// TIA Portal V15.1 export
// export: Created 2024-05-17T05:38:39.8401583Z, ExportSetting WithDefaults, DisplayName Totally Integrated Automation Portal, DisplayVersion V15.1 Update 5, DisplayName TIA Portal Openness, DisplayVersion V15.1 Update 5, DisplayName SINAMICS Startdrive Advanced, DisplayVersion V15.1, DisplayName G130, G150, S120, S150, SINAMICS MV, S210, DisplayVersion V15.1, DisplayName G110M, G120, G120C, G120D, G120P, DisplayVersion V15.1, DisplayName STEP 7 Professional, DisplayVersion V15.1 Update 5, DisplayName STEP 7 Safety, DisplayVersion V15.1, DisplayName WinCC Professional, DisplayVersion V15.1 Update 5, DisplayName SIMATIC Visualization Architect, DisplayVersion V15.1
FUNCTION_BLOCK "LGBBitShift"   // FB6690, FBD
TITLE = LGBBitShift
{ S7_Optimized_Access := 'TRUE' }
VERSION : 0.1
// stored: AutoNumber false, IsIECCheckEnabled false, IsRetainMemResEnabled false, MemoryReserve 100, SetENOAutomatically False, UDAEnableTagReadback false
   VAR_INPUT
      I_ArrivedToPrev1 { ExternalAccessible := 'False'; ExternalVisible := 'False'; ExternalWritable := 'False'} : Bool;   // Arrived signal to previous transfer 1
      I_Bits1 { ExternalAccessible := 'False'; ExternalVisible := 'False'; ExternalWritable := 'False'} : Word;   // Bits transfer 1
      I_ArrivedToPrev2 { ExternalAccessible := 'False'; ExternalVisible := 'False'; ExternalWritable := 'False'} : Bool;   // Arrived signal to previous transfer 2
      I_Bits2 { ExternalAccessible := 'False'; ExternalVisible := 'False'; ExternalWritable := 'False'} : Word;   // Bits transfer 2
      I_ArrivedToPrev3 { ExternalAccessible := 'False'; ExternalVisible := 'False'; ExternalWritable := 'False'} : Bool;   // Arrived signal to previous transfer 3
      I_Bits3 { ExternalAccessible := 'False'; ExternalVisible := 'False'; ExternalWritable := 'False'} : Word;   // Bits transfer 3
      I_ArrivedToPrev4 { ExternalAccessible := 'False'; ExternalVisible := 'False'; ExternalWritable := 'False'} : Bool;   // Arrived signal to previous transfer 4
      I_Bits4 { ExternalAccessible := 'False'; ExternalVisible := 'False'; ExternalWritable := 'False'} : Word;   // Bits transfer 4
      I_NextShiftDone { ExternalAccessible := 'False'; ExternalVisible := 'False'; ExternalWritable := 'False'} : Bool;   // Shift to next position is done
   END_VAR
   VAR_OUTPUT
      O_ShiftDone1 { ExternalAccessible := 'False'; ExternalVisible := 'False'; ExternalWritable := 'False'} : Bool;   // Shift done transfer 1
      O_ShiftDone2 { ExternalAccessible := 'False'; ExternalVisible := 'False'; ExternalWritable := 'False'} : Bool;   // Shift done transfer 2
      O_ShiftDone3 { ExternalAccessible := 'False'; ExternalVisible := 'False'; ExternalWritable := 'False'} : Bool;   // Shift done transfer 3
      O_ShiftDone4 { ExternalAccessible := 'False'; ExternalVisible := 'False'; ExternalWritable := 'False'} : Bool;   // Shift done transfer 4
      O_Bits { ExternalAccessible := 'False'; ExternalVisible := 'False'; ExternalWritable := 'False'} : Int;   // Bits for this position
      O_Bit0 { ExternalAccessible := 'False'; ExternalVisible := 'False'; ExternalWritable := 'False'} : Bool;   // Bit 0
      O_Bit1 { ExternalAccessible := 'False'; ExternalVisible := 'False'; ExternalWritable := 'False'} : Bool;   // Bit 1
      O_Bit2 { ExternalAccessible := 'False'; ExternalVisible := 'False'; ExternalWritable := 'False'} : Bool;   // Bit 2
      O_Bit3 { ExternalAccessible := 'False'; ExternalVisible := 'False'; ExternalWritable := 'False'} : Bool;   // Bit 3
      O_Bit4 { ExternalAccessible := 'False'; ExternalVisible := 'False'; ExternalWritable := 'False'} : Bool;   // Bit 4
      O_Bit5 { ExternalAccessible := 'False'; ExternalVisible := 'False'; ExternalWritable := 'False'} : Bool;   // Bit 5
      O_Bit6 { ExternalAccessible := 'False'; ExternalVisible := 'False'; ExternalWritable := 'False'} : Bool;   // Bit 6
      O_Bit7 { ExternalAccessible := 'False'; ExternalVisible := 'False'; ExternalWritable := 'False'} : Bool;   // Bit 7
      O_Bit8 { ExternalAccessible := 'False'; ExternalVisible := 'False'; ExternalWritable := 'False'} : Bool;   // Bit 8
      O_Bit9 { ExternalAccessible := 'False'; ExternalVisible := 'False'; ExternalWritable := 'False'} : Bool;   // Bit 9
      O_Bit10 { ExternalAccessible := 'False'; ExternalVisible := 'False'; ExternalWritable := 'False'} : Bool;   // Bit 10
      O_Bit11 { ExternalAccessible := 'False'; ExternalVisible := 'False'; ExternalWritable := 'False'} : Bool;   // Bit 11
      O_Bit12 { ExternalAccessible := 'False'; ExternalVisible := 'False'; ExternalWritable := 'False'} : Bool;   // Bit 12
      O_Bit13 { ExternalAccessible := 'False'; ExternalVisible := 'False'; ExternalWritable := 'False'} : Bool;   // Bit 13
      O_Bit14 { ExternalAccessible := 'False'; ExternalVisible := 'False'; ExternalWritable := 'False'} : Bool;   // Bit 14
      O_Bit15 { ExternalAccessible := 'False'; ExternalVisible := 'False'; ExternalWritable := 'False'} : Bool;   // Bit 15
      O_AlarmABCondition { ExternalAccessible := 'False'; ExternalVisible := 'False'; ExternalWritable := 'False'} : Bool;   // Alarm AB Condition
      O_AlarmA { ExternalAccessible := 'False'; ExternalVisible := 'False'; ExternalWritable := 'False'} : Bool;   // Alarm A
      O_AlarmB { ExternalAccessible := 'False'; ExternalVisible := 'False'; ExternalWritable := 'False'} : Bool;   // Alarm B
      O_AlarmC { ExternalAccessible := 'False'; ExternalVisible := 'False'; ExternalWritable := 'False'} : Bool;   // Alarm C
      O_AlarmD { ExternalAccessible := 'False'; ExternalVisible := 'False'; ExternalWritable := 'False'} : Bool;   // Alarm D
      H_AlarmDWord { ExternalAccessible := 'False'; ExternalVisible := 'False'; ExternalWritable := 'False'} : DWord;   // HMI Animation
   END_VAR
   VAR_IN_OUT
      IO_Modes : "Modes";   // Modes
      H_HMI : "H_HMI";   // Icon Animation
      H_GBBitShift : "H_GBBitShift";   // Animation
      C_Config : "BitShiftConfig";   // Config
   END_VAR
   VAR
      AC_NoBitShift { ExternalAccessible := 'False'; ExternalVisible := 'False'; ExternalWritable := 'False'} : Bool;   // Alarm No Bit Shift
      PulseArrivedToPrev1 { ExternalAccessible := 'False'; ExternalVisible := 'False'; ExternalWritable := 'False'} : Bool;   // Pulse Arrived Signal to Previous Transfer 1
      Arrived1 { ExternalAccessible := 'False'; ExternalVisible := 'False'; ExternalWritable := 'False'} : Bool;   // Arrived 1
      PulseArrivedToPrev2 { ExternalAccessible := 'False'; ExternalVisible := 'False'; ExternalWritable := 'False'} : Bool;   // Pulse Arrived Signal to Previous Transfer 2
      Arrived2 { ExternalAccessible := 'False'; ExternalVisible := 'False'; ExternalWritable := 'False'} : Bool;   // Arrived 2
      PulseArrivedToPrev3 { ExternalAccessible := 'False'; ExternalVisible := 'False'; ExternalWritable := 'False'} : Bool;   // Pulse Arrived Signal to Previous Transfer 3
      Arrived3 { ExternalAccessible := 'False'; ExternalVisible := 'False'; ExternalWritable := 'False'} : Bool;   // Arrived 3
      PulseArrivedToPrev4 { ExternalAccessible := 'False'; ExternalVisible := 'False'; ExternalWritable := 'False'} : Bool;   // Pulse Arrived Signal to Previous Transfer 4
      Arrived4 { ExternalAccessible := 'False'; ExternalVisible := 'False'; ExternalWritable := 'False'} : Bool;   // Arrived 4
   END_VAR
   VAR RETAIN
      Bits { ExternalAccessible := 'False'; ExternalVisible := 'False'; ExternalWritable := 'False'} : Word;   // Bits of this position
   END_VAR
   VAR
      AlarmA { ExternalAccessible := 'False'; ExternalVisible := 'False'; ExternalWritable := 'False'} : Bool;   // Alarm A
      AlarmB { ExternalAccessible := 'False'; ExternalVisible := 'False'; ExternalWritable := 'False'} : Bool;   // Alarm B
      AlarmC { ExternalAccessible := 'False'; ExternalVisible := 'False'; ExternalWritable := 'False'} : Bool;   // Alarm C
      AlarmD { ExternalAccessible := 'False'; ExternalVisible := 'False'; ExternalWritable := 'False'} : Bool;   // Alarm D
      AlarmABCondition { ExternalAccessible := 'False'; ExternalVisible := 'False'; ExternalWritable := 'False'} : Bool;   // Alarm AB Condition
   END_VAR
   VAR_TEMP   // added for the SCL form of the ladder/FBD networks
      _w1 : Bool;
   END_VAR
BEGIN

REGION Network 1: **** 4.4 - Machine status - Calculated **** Pulse Arrived Signal 1 To previous
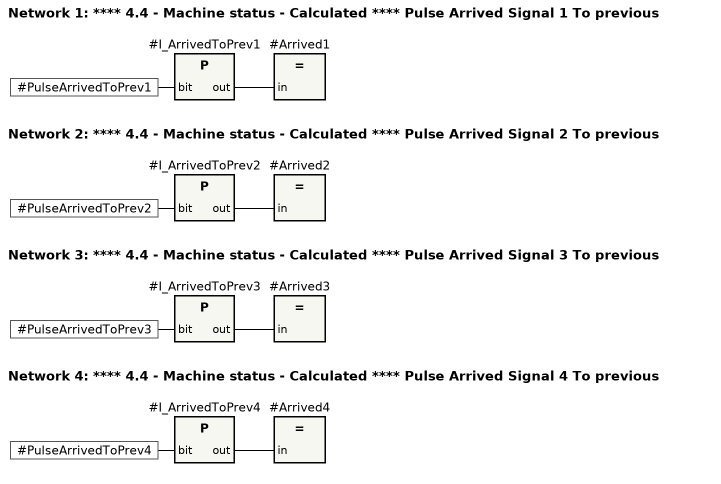
   #_w1 := #I_ArrivedToPrev1 AND NOT #PulseArrivedToPrev1;   // rising edge of #I_ArrivedToPrev1
   #PulseArrivedToPrev1 := #I_ArrivedToPrev1;
   #Arrived1 := #_w1;
END_REGION

REGION Network 2: **** 4.4 - Machine status - Calculated **** Pulse Arrived Signal 2 To previous
   #_w1 := #I_ArrivedToPrev2 AND NOT #PulseArrivedToPrev2;   // rising edge of #I_ArrivedToPrev2
   #PulseArrivedToPrev2 := #I_ArrivedToPrev2;
   #Arrived2 := #_w1;
END_REGION

REGION Network 3: **** 4.4 - Machine status - Calculated **** Pulse Arrived Signal 3 To previous
   #_w1 := #I_ArrivedToPrev3 AND NOT #PulseArrivedToPrev3;   // rising edge of #I_ArrivedToPrev3
   #PulseArrivedToPrev3 := #I_ArrivedToPrev3;
   #Arrived3 := #_w1;
END_REGION

REGION Network 4: **** 4.4 - Machine status - Calculated **** Pulse Arrived Signal 4 To previous
   #_w1 := #I_ArrivedToPrev4 AND NOT #PulseArrivedToPrev4;   // rising edge of #I_ArrivedToPrev4
   #PulseArrivedToPrev4 := #I_ArrivedToPrev4;
   #Arrived4 := #_w1;
END_REGION

REGION Network 5: **** 4.4 - Machine status - Calculated **** Copy Bits from Transfer 1
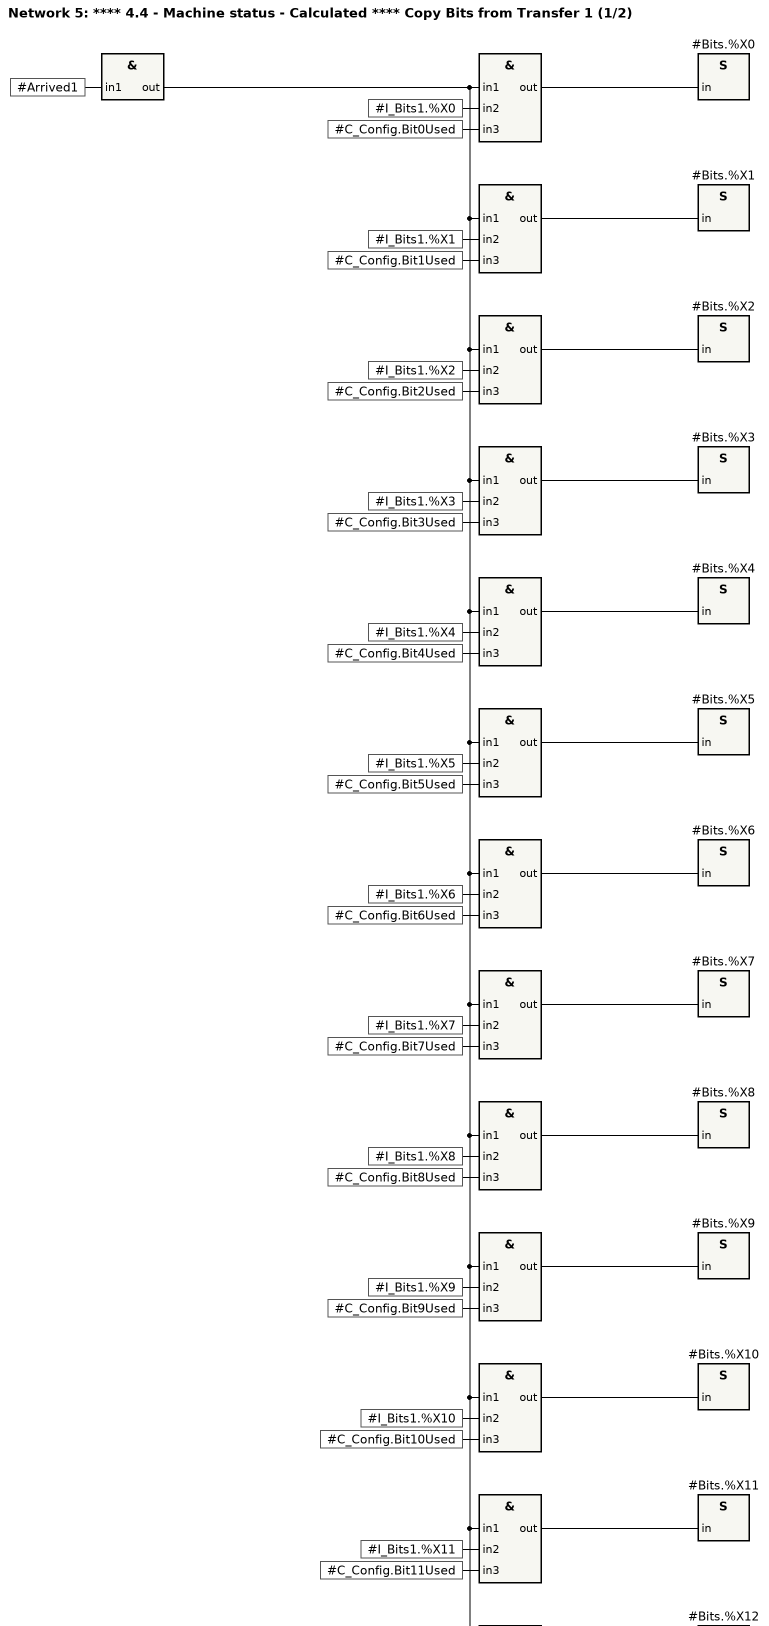
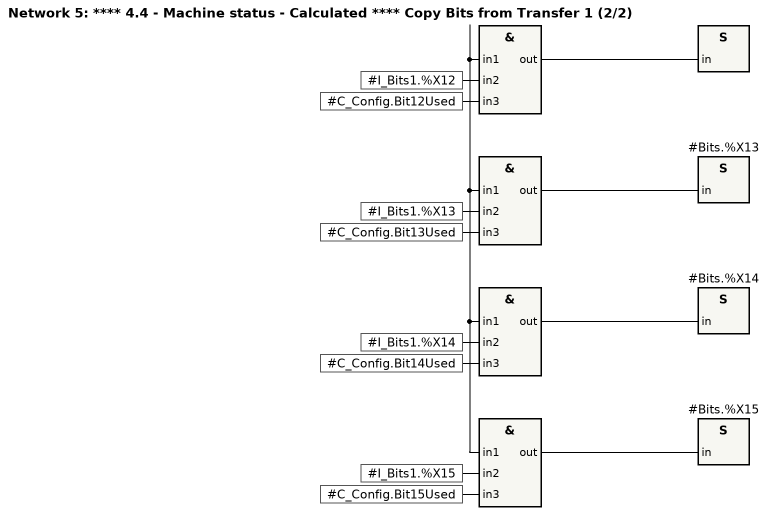
   IF #Arrived1 AND #I_Bits1.%X0 AND #C_Config.Bit0Used THEN #Bits.%X0 := TRUE; END_IF;
   IF #Arrived1 AND #I_Bits1.%X1 AND #C_Config.Bit1Used THEN #Bits.%X1 := TRUE; END_IF;
   IF #Arrived1 AND #I_Bits1.%X2 AND #C_Config.Bit2Used THEN #Bits.%X2 := TRUE; END_IF;
   IF #Arrived1 AND #I_Bits1.%X3 AND #C_Config.Bit3Used THEN #Bits.%X3 := TRUE; END_IF;
   IF #Arrived1 AND #I_Bits1.%X4 AND #C_Config.Bit4Used THEN #Bits.%X4 := TRUE; END_IF;
   IF #Arrived1 AND #I_Bits1.%X5 AND #C_Config.Bit5Used THEN #Bits.%X5 := TRUE; END_IF;
   IF #Arrived1 AND #I_Bits1.%X6 AND #C_Config.Bit6Used THEN #Bits.%X6 := TRUE; END_IF;
   IF #Arrived1 AND #I_Bits1.%X7 AND #C_Config.Bit7Used THEN #Bits.%X7 := TRUE; END_IF;
   IF #Arrived1 AND #I_Bits1.%X8 AND #C_Config.Bit8Used THEN #Bits.%X8 := TRUE; END_IF;
   IF #Arrived1 AND #I_Bits1.%X9 AND #C_Config.Bit9Used THEN #Bits.%X9 := TRUE; END_IF;
   IF #Arrived1 AND #I_Bits1.%X10 AND #C_Config.Bit10Used THEN #Bits.%X10 := TRUE; END_IF;
   IF #Arrived1 AND #I_Bits1.%X11 AND #C_Config.Bit11Used THEN #Bits.%X11 := TRUE; END_IF;
   IF #Arrived1 AND #I_Bits1.%X12 AND #C_Config.Bit12Used THEN #Bits.%X12 := TRUE; END_IF;
   IF #Arrived1 AND #I_Bits1.%X13 AND #C_Config.Bit13Used THEN #Bits.%X13 := TRUE; END_IF;
   IF #Arrived1 AND #I_Bits1.%X14 AND #C_Config.Bit14Used THEN #Bits.%X14 := TRUE; END_IF;
   IF #Arrived1 AND #I_Bits1.%X15 AND #C_Config.Bit15Used THEN #Bits.%X15 := TRUE; END_IF;
END_REGION

REGION Network 6: **** 4.4 - Machine status - Calculated **** Copy Bits from Transfer 2
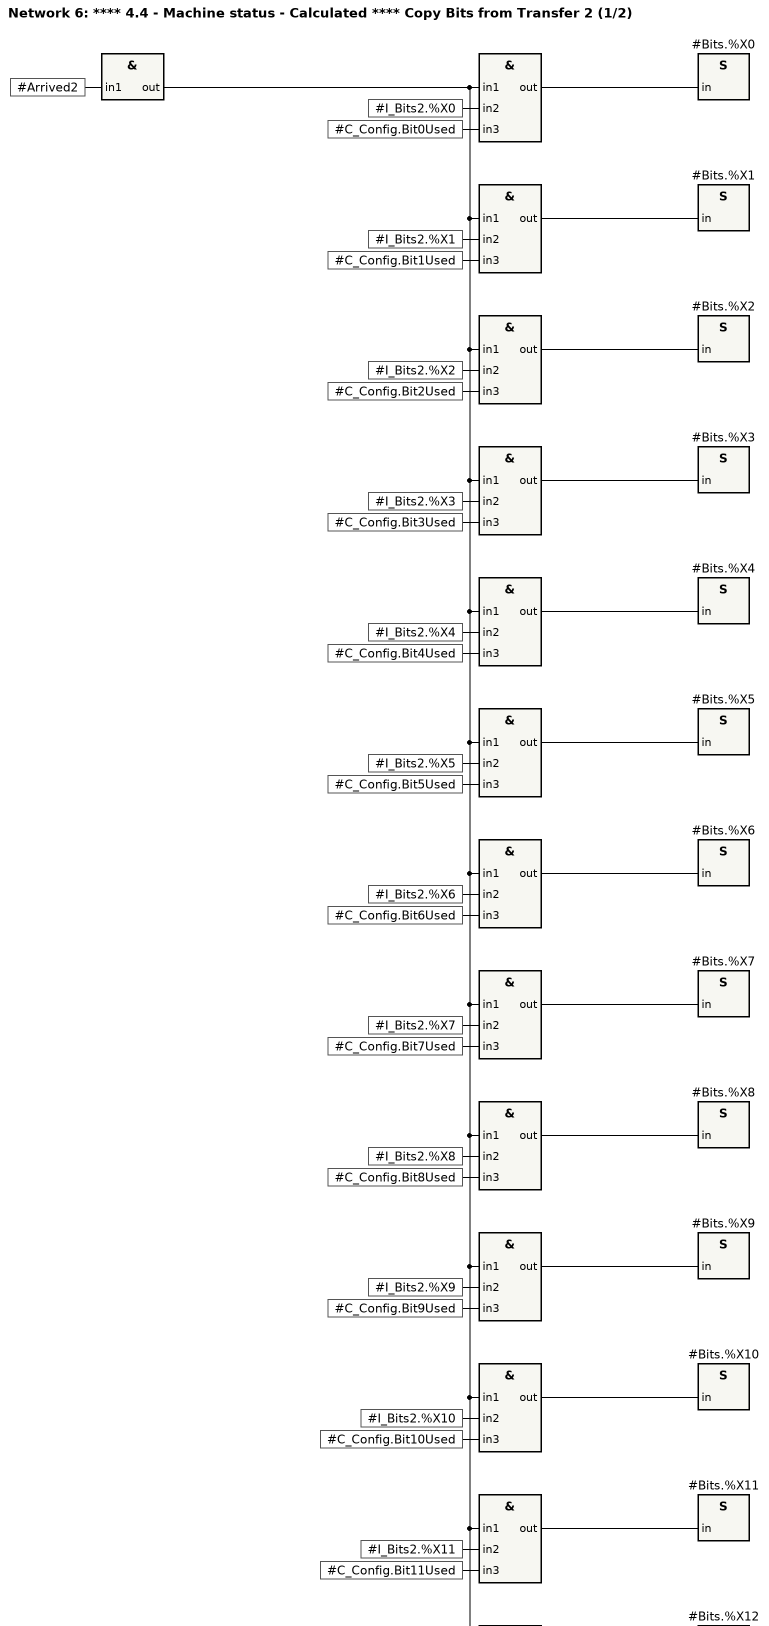
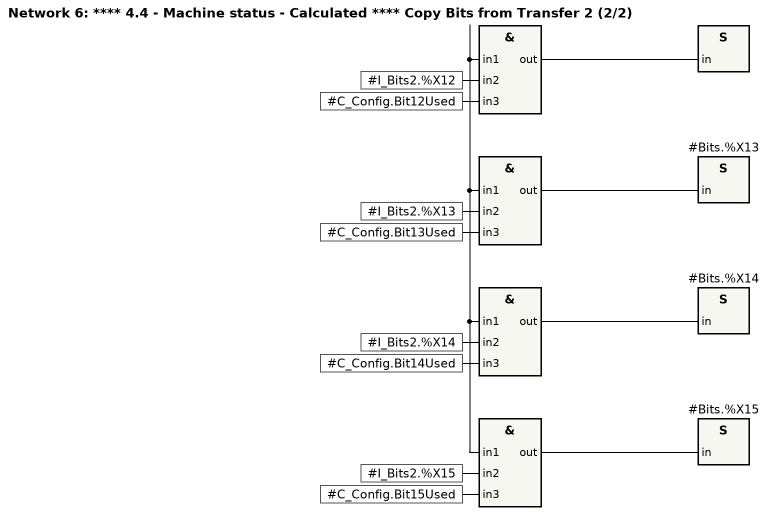
   IF #Arrived2 AND #I_Bits2.%X0 AND #C_Config.Bit0Used THEN #Bits.%X0 := TRUE; END_IF;
   IF #Arrived2 AND #I_Bits2.%X1 AND #C_Config.Bit1Used THEN #Bits.%X1 := TRUE; END_IF;
   IF #Arrived2 AND #I_Bits2.%X2 AND #C_Config.Bit2Used THEN #Bits.%X2 := TRUE; END_IF;
   IF #Arrived2 AND #I_Bits2.%X3 AND #C_Config.Bit3Used THEN #Bits.%X3 := TRUE; END_IF;
   IF #Arrived2 AND #I_Bits2.%X4 AND #C_Config.Bit4Used THEN #Bits.%X4 := TRUE; END_IF;
   IF #Arrived2 AND #I_Bits2.%X5 AND #C_Config.Bit5Used THEN #Bits.%X5 := TRUE; END_IF;
   IF #Arrived2 AND #I_Bits2.%X6 AND #C_Config.Bit6Used THEN #Bits.%X6 := TRUE; END_IF;
   IF #Arrived2 AND #I_Bits2.%X7 AND #C_Config.Bit7Used THEN #Bits.%X7 := TRUE; END_IF;
   IF #Arrived2 AND #I_Bits2.%X8 AND #C_Config.Bit8Used THEN #Bits.%X8 := TRUE; END_IF;
   IF #Arrived2 AND #I_Bits2.%X9 AND #C_Config.Bit9Used THEN #Bits.%X9 := TRUE; END_IF;
   IF #Arrived2 AND #I_Bits2.%X10 AND #C_Config.Bit10Used THEN #Bits.%X10 := TRUE; END_IF;
   IF #Arrived2 AND #I_Bits2.%X11 AND #C_Config.Bit11Used THEN #Bits.%X11 := TRUE; END_IF;
   IF #Arrived2 AND #I_Bits2.%X12 AND #C_Config.Bit12Used THEN #Bits.%X12 := TRUE; END_IF;
   IF #Arrived2 AND #I_Bits2.%X13 AND #C_Config.Bit13Used THEN #Bits.%X13 := TRUE; END_IF;
   IF #Arrived2 AND #I_Bits2.%X14 AND #C_Config.Bit14Used THEN #Bits.%X14 := TRUE; END_IF;
   IF #Arrived2 AND #I_Bits2.%X15 AND #C_Config.Bit15Used THEN #Bits.%X15 := TRUE; END_IF;
END_REGION

REGION Network 7: **** 4.4 - Machine status - Calculated **** Copy Bits from Transfer 3
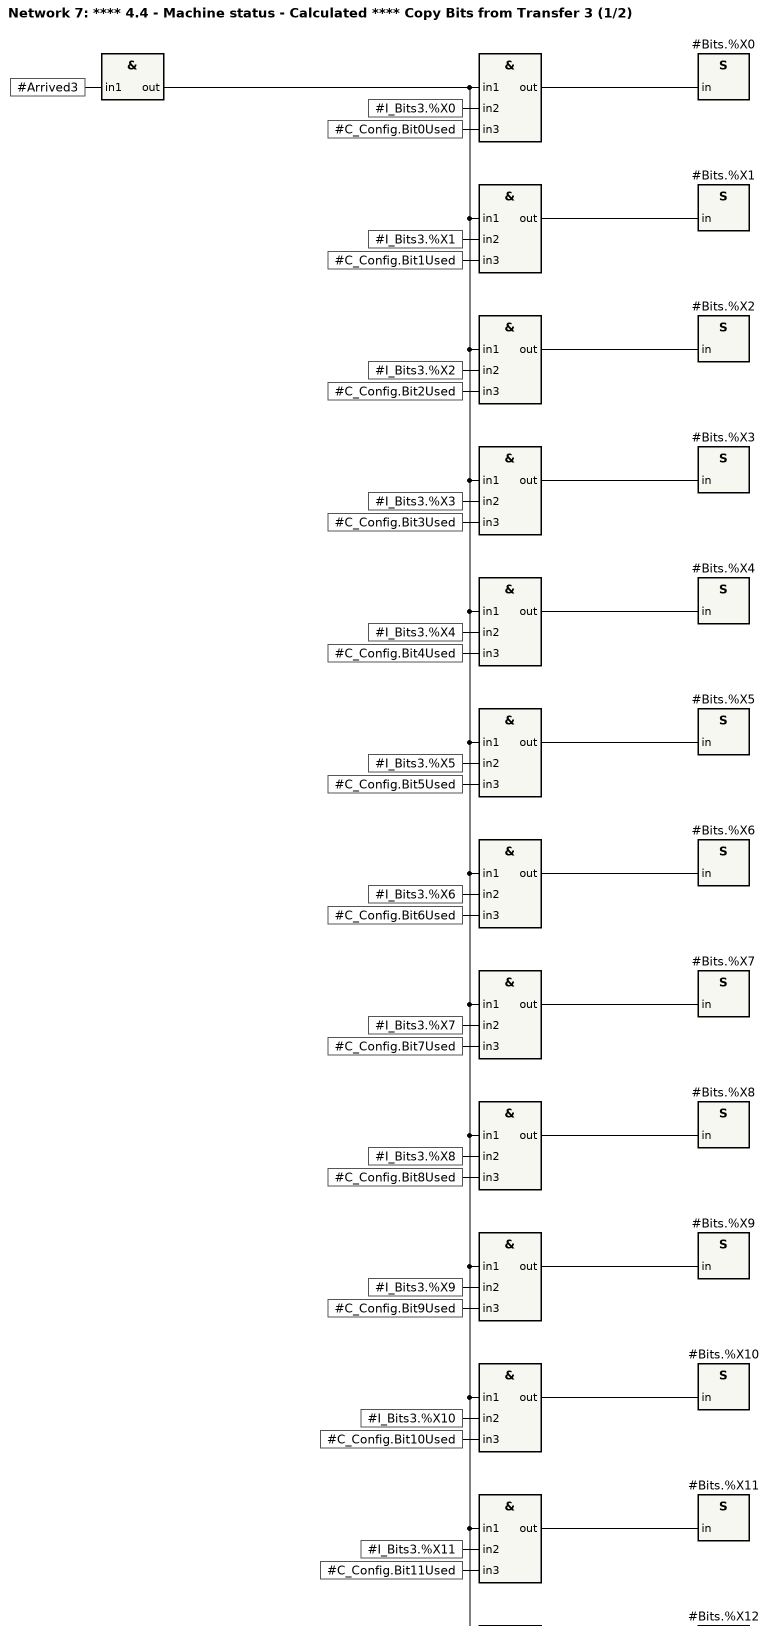
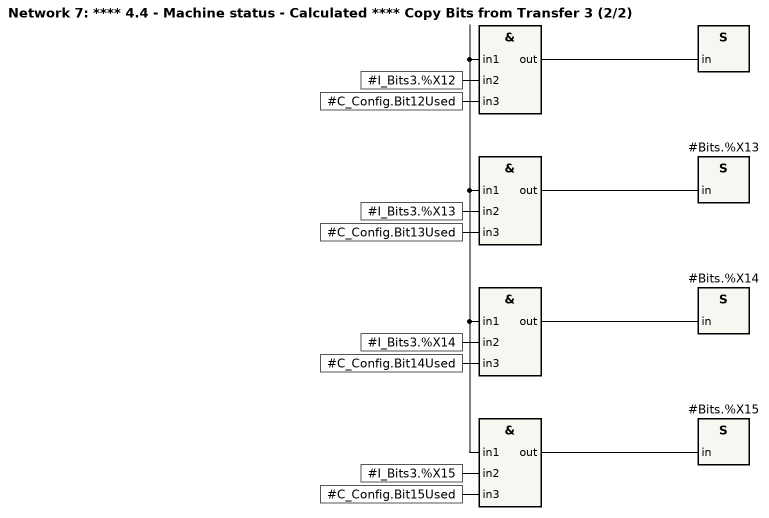
   IF #Arrived3 AND #I_Bits3.%X0 AND #C_Config.Bit0Used THEN #Bits.%X0 := TRUE; END_IF;
   IF #Arrived3 AND #I_Bits3.%X1 AND #C_Config.Bit1Used THEN #Bits.%X1 := TRUE; END_IF;
   IF #Arrived3 AND #I_Bits3.%X2 AND #C_Config.Bit2Used THEN #Bits.%X2 := TRUE; END_IF;
   IF #Arrived3 AND #I_Bits3.%X3 AND #C_Config.Bit3Used THEN #Bits.%X3 := TRUE; END_IF;
   IF #Arrived3 AND #I_Bits3.%X4 AND #C_Config.Bit4Used THEN #Bits.%X4 := TRUE; END_IF;
   IF #Arrived3 AND #I_Bits3.%X5 AND #C_Config.Bit5Used THEN #Bits.%X5 := TRUE; END_IF;
   IF #Arrived3 AND #I_Bits3.%X6 AND #C_Config.Bit6Used THEN #Bits.%X6 := TRUE; END_IF;
   IF #Arrived3 AND #I_Bits3.%X7 AND #C_Config.Bit7Used THEN #Bits.%X7 := TRUE; END_IF;
   IF #Arrived3 AND #I_Bits3.%X8 AND #C_Config.Bit8Used THEN #Bits.%X8 := TRUE; END_IF;
   IF #Arrived3 AND #I_Bits3.%X9 AND #C_Config.Bit9Used THEN #Bits.%X9 := TRUE; END_IF;
   IF #Arrived3 AND #I_Bits3.%X10 AND #C_Config.Bit10Used THEN #Bits.%X10 := TRUE; END_IF;
   IF #Arrived3 AND #I_Bits3.%X11 AND #C_Config.Bit11Used THEN #Bits.%X11 := TRUE; END_IF;
   IF #Arrived3 AND #I_Bits3.%X12 AND #C_Config.Bit12Used THEN #Bits.%X12 := TRUE; END_IF;
   IF #Arrived3 AND #I_Bits3.%X13 AND #C_Config.Bit13Used THEN #Bits.%X13 := TRUE; END_IF;
   IF #Arrived3 AND #I_Bits3.%X14 AND #C_Config.Bit14Used THEN #Bits.%X14 := TRUE; END_IF;
   IF #Arrived3 AND #I_Bits3.%X15 AND #C_Config.Bit15Used THEN #Bits.%X15 := TRUE; END_IF;
END_REGION

REGION Network 8: **** 4.4 - Machine status - Calculated **** Copy Bits from Transfer 4
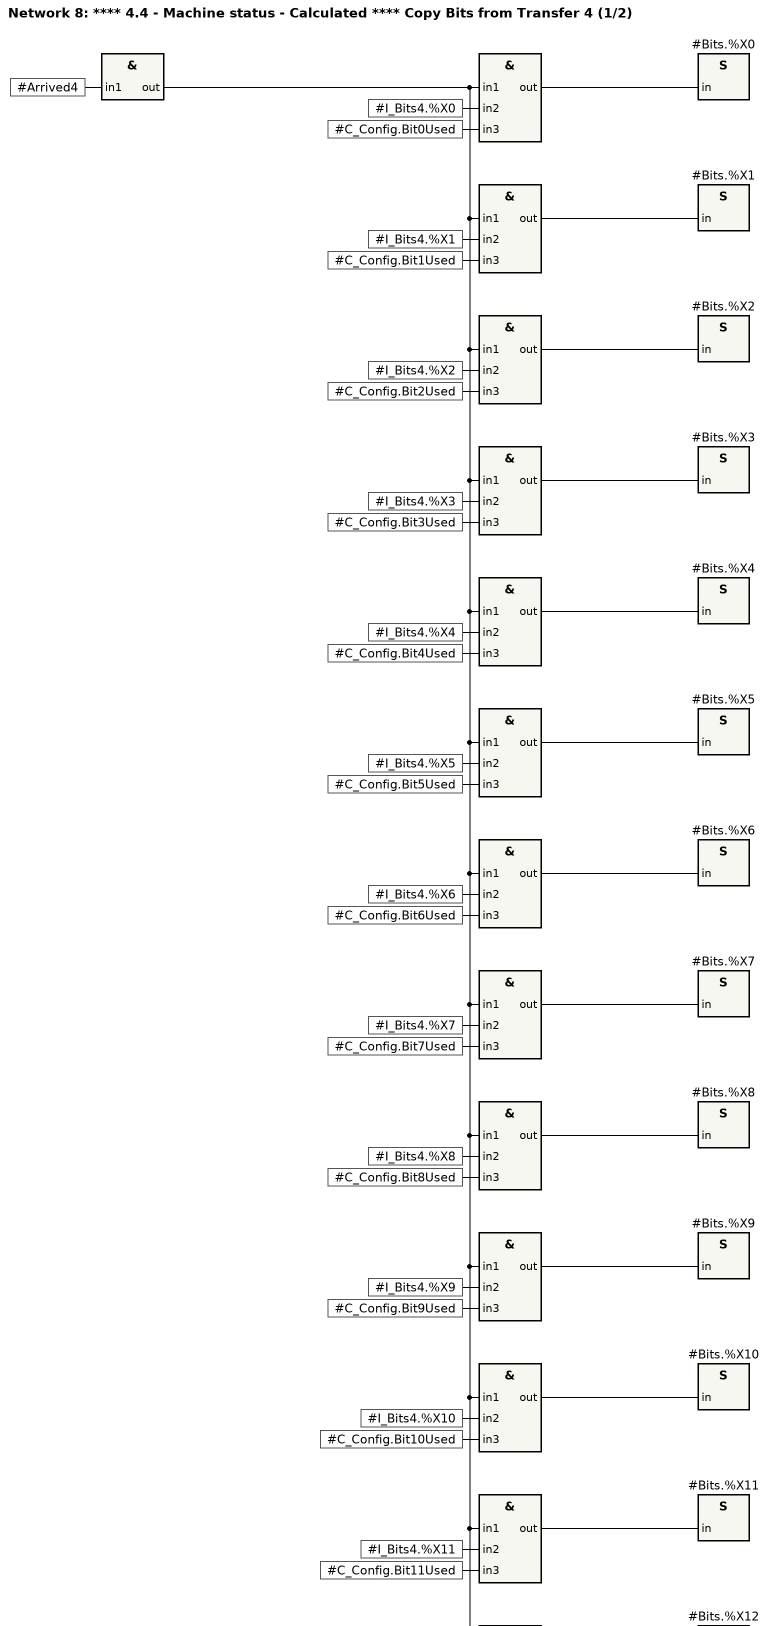
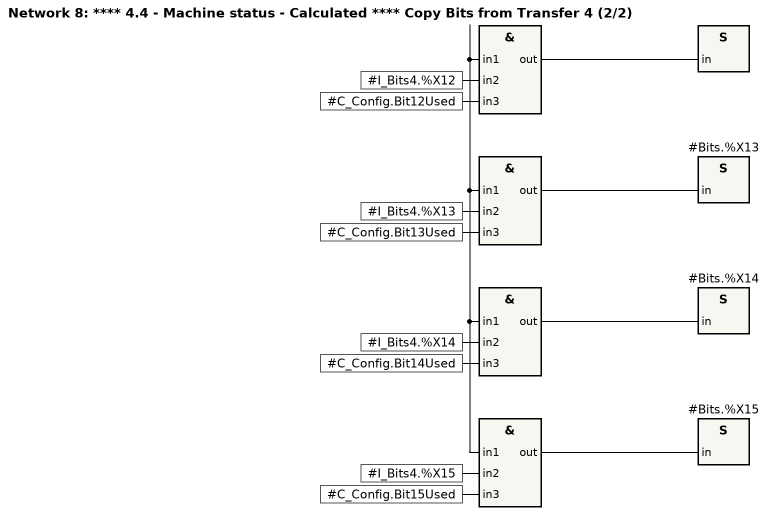
   IF #Arrived4 AND #I_Bits4.%X0 AND #C_Config.Bit0Used THEN #Bits.%X0 := TRUE; END_IF;
   IF #Arrived4 AND #I_Bits4.%X1 AND #C_Config.Bit1Used THEN #Bits.%X1 := TRUE; END_IF;
   IF #Arrived4 AND #I_Bits4.%X2 AND #C_Config.Bit2Used THEN #Bits.%X2 := TRUE; END_IF;
   IF #Arrived4 AND #I_Bits4.%X3 AND #C_Config.Bit3Used THEN #Bits.%X3 := TRUE; END_IF;
   IF #Arrived4 AND #I_Bits4.%X4 AND #C_Config.Bit4Used THEN #Bits.%X4 := TRUE; END_IF;
   IF #Arrived4 AND #I_Bits4.%X5 AND #C_Config.Bit5Used THEN #Bits.%X5 := TRUE; END_IF;
   IF #Arrived4 AND #I_Bits4.%X6 AND #C_Config.Bit6Used THEN #Bits.%X6 := TRUE; END_IF;
   IF #Arrived4 AND #I_Bits4.%X7 AND #C_Config.Bit7Used THEN #Bits.%X7 := TRUE; END_IF;
   IF #Arrived4 AND #I_Bits4.%X8 AND #C_Config.Bit8Used THEN #Bits.%X8 := TRUE; END_IF;
   IF #Arrived4 AND #I_Bits4.%X9 AND #C_Config.Bit9Used THEN #Bits.%X9 := TRUE; END_IF;
   IF #Arrived4 AND #I_Bits4.%X10 AND #C_Config.Bit10Used THEN #Bits.%X10 := TRUE; END_IF;
   IF #Arrived4 AND #I_Bits4.%X11 AND #C_Config.Bit11Used THEN #Bits.%X11 := TRUE; END_IF;
   IF #Arrived4 AND #I_Bits4.%X12 AND #C_Config.Bit12Used THEN #Bits.%X12 := TRUE; END_IF;
   IF #Arrived4 AND #I_Bits4.%X13 AND #C_Config.Bit13Used THEN #Bits.%X13 := TRUE; END_IF;
   IF #Arrived4 AND #I_Bits4.%X14 AND #C_Config.Bit14Used THEN #Bits.%X14 := TRUE; END_IF;
   IF #Arrived4 AND #I_Bits4.%X15 AND #C_Config.Bit15Used THEN #Bits.%X15 := TRUE; END_IF;
END_REGION

REGION Network 9: **** 4.4 - Machine status - Calculated **** Reset Data when shift to the next position is done
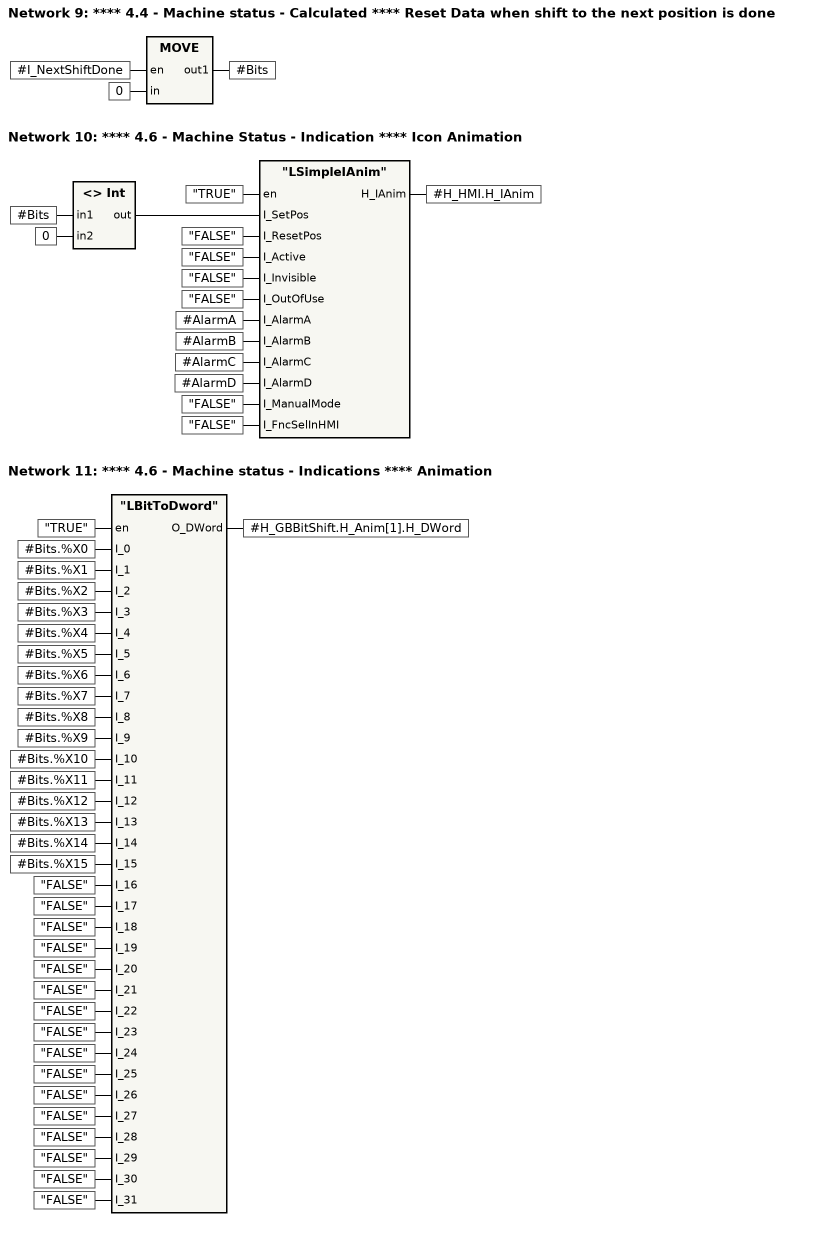
   IF #I_NextShiftDone THEN #Bits := 0; END_IF;
END_REGION

REGION Network 10: **** 4.6 - Machine Status - Indication **** Icon Animation
   IF "TRUE" THEN
       "LSimpleIAnim"(I_SetPos := #Bits <> 0,
                      I_ResetPos := "FALSE",
                      I_Active := "FALSE",
                      I_Invisible := "FALSE",
                      I_OutOfUse := "FALSE",
                      I_AlarmA := #AlarmA,
                      I_AlarmB := #AlarmB,
                      I_AlarmC := #AlarmC,
                      I_AlarmD := #AlarmD,
                      I_ManualMode := "FALSE",
                      I_FncSelInHMI := "FALSE",
                      H_IAnim => #H_HMI.H_IAnim);
   END_IF;
END_REGION

REGION Network 11: **** 4.6 - Machine status - Indications **** Animation
   IF "TRUE" THEN
       "LBitToDword"(I_0 := #Bits.%X0,
                     I_1 := #Bits.%X1,
                     I_2 := #Bits.%X2,
                     I_3 := #Bits.%X3,
                     I_4 := #Bits.%X4,
                     I_5 := #Bits.%X5,
                     I_6 := #Bits.%X6,
                     I_7 := #Bits.%X7,
                     I_8 := #Bits.%X8,
                     I_9 := #Bits.%X9,
                     I_10 := #Bits.%X10,
                     I_11 := #Bits.%X11,
                     I_12 := #Bits.%X12,
                     I_13 := #Bits.%X13,
                     I_14 := #Bits.%X14,
                     I_15 := #Bits.%X15,
                     I_16 := "FALSE",
                     I_17 := "FALSE",
                     I_18 := "FALSE",
                     I_19 := "FALSE",
                     I_20 := "FALSE",
                     I_21 := "FALSE",
                     I_22 := "FALSE",
                     I_23 := "FALSE",
                     I_24 := "FALSE",
                     I_25 := "FALSE",
                     I_26 := "FALSE",
                     I_27 := "FALSE",
                     I_28 := "FALSE",
                     I_29 := "FALSE",
                     I_30 := "FALSE",
                     I_31 := "FALSE",
                     O_DWord => #H_GBBitShift.H_Anim[1].H_DWord);
   END_IF;
END_REGION

REGION Network 12: **** 4.6 - Machine status - Indications **** Animation
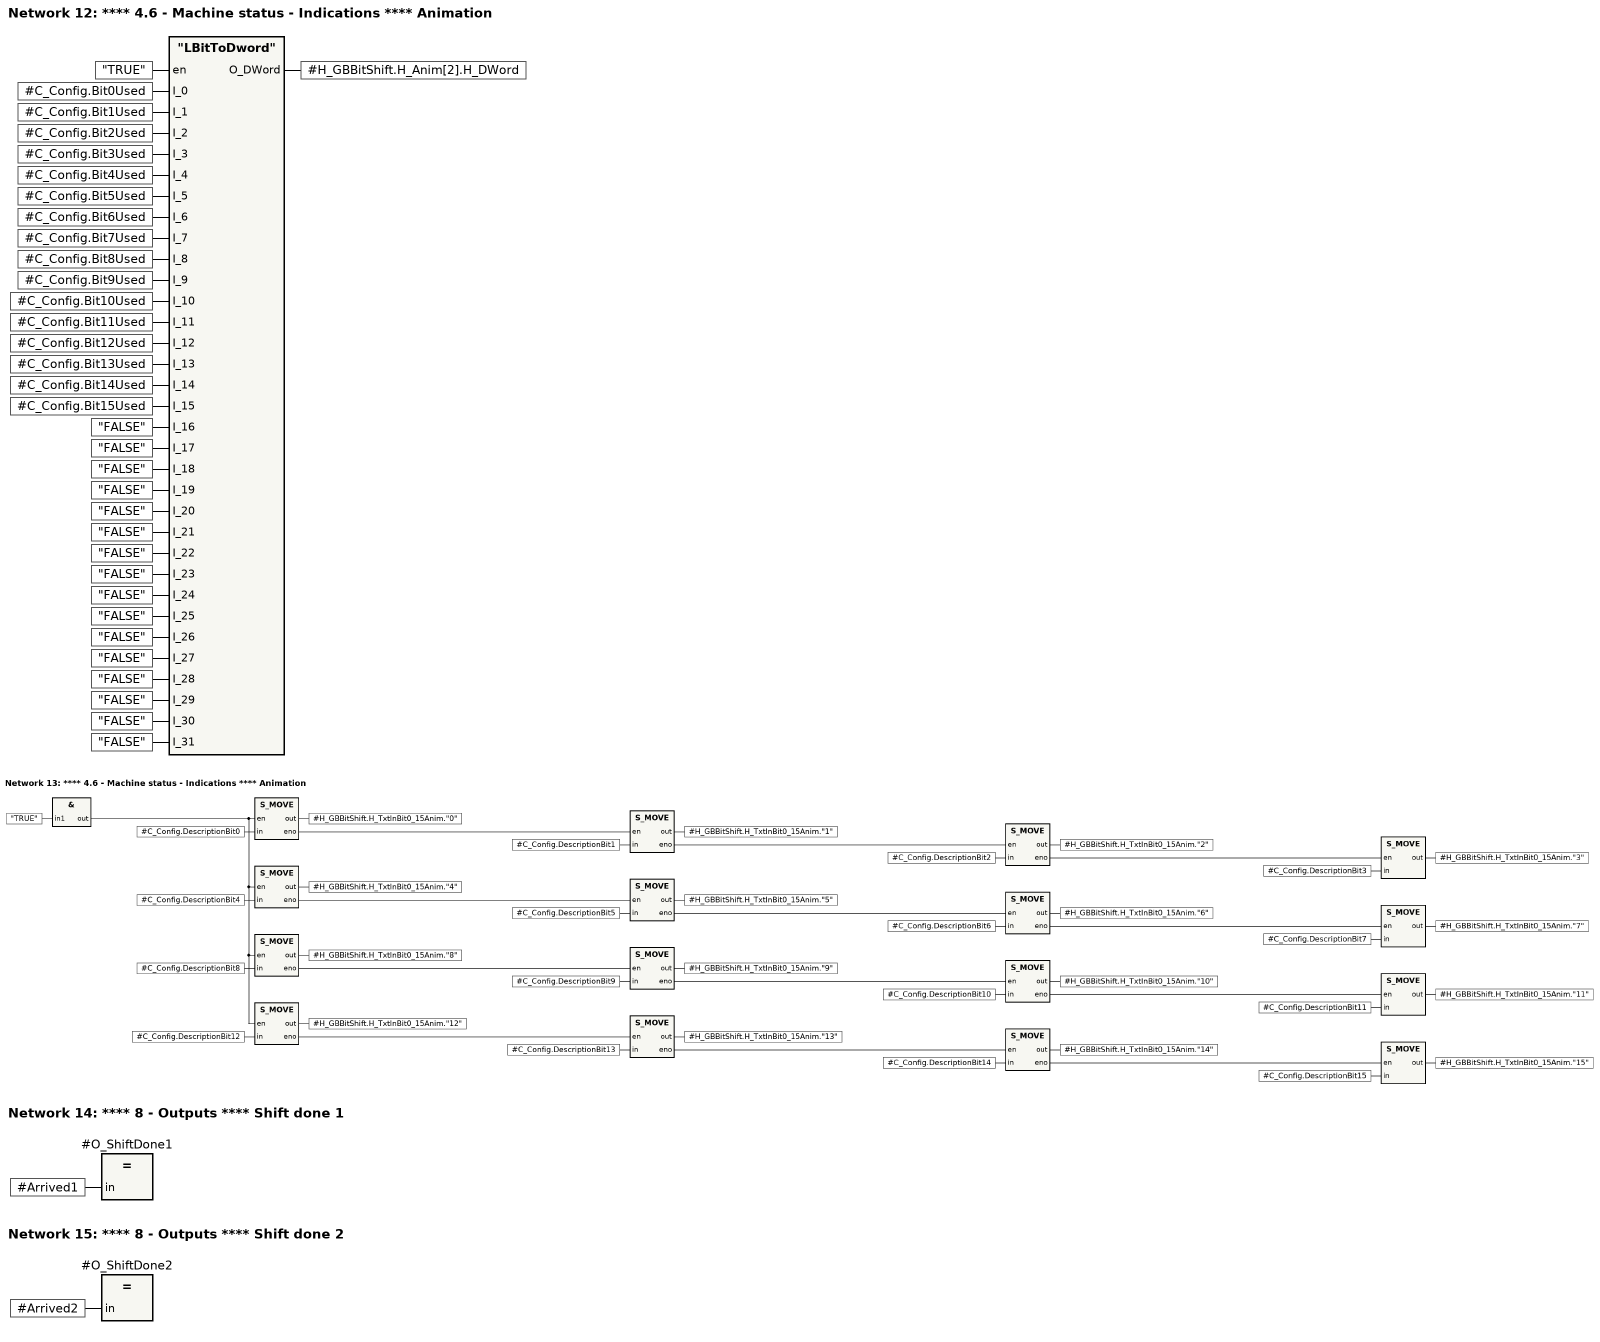
   IF "TRUE" THEN
       "LBitToDword"(I_0 := #C_Config.Bit0Used,
                     I_1 := #C_Config.Bit1Used,
                     I_2 := #C_Config.Bit2Used,
                     I_3 := #C_Config.Bit3Used,
                     I_4 := #C_Config.Bit4Used,
                     I_5 := #C_Config.Bit5Used,
                     I_6 := #C_Config.Bit6Used,
                     I_7 := #C_Config.Bit7Used,
                     I_8 := #C_Config.Bit8Used,
                     I_9 := #C_Config.Bit9Used,
                     I_10 := #C_Config.Bit10Used,
                     I_11 := #C_Config.Bit11Used,
                     I_12 := #C_Config.Bit12Used,
                     I_13 := #C_Config.Bit13Used,
                     I_14 := #C_Config.Bit14Used,
                     I_15 := #C_Config.Bit15Used,
                     I_16 := "FALSE",
                     I_17 := "FALSE",
                     I_18 := "FALSE",
                     I_19 := "FALSE",
                     I_20 := "FALSE",
                     I_21 := "FALSE",
                     I_22 := "FALSE",
                     I_23 := "FALSE",
                     I_24 := "FALSE",
                     I_25 := "FALSE",
                     I_26 := "FALSE",
                     I_27 := "FALSE",
                     I_28 := "FALSE",
                     I_29 := "FALSE",
                     I_30 := "FALSE",
                     I_31 := "FALSE",
                     O_DWord => #H_GBBitShift.H_Anim[2].H_DWord);
   END_IF;
END_REGION

REGION Network 13: **** 4.6 - Machine status - Indications **** Animation
   IF "TRUE" THEN
       #H_GBBitShift.H_TxtInBit0_15Anim."0" := #C_Config.DescriptionBit0;
       #H_GBBitShift.H_TxtInBit0_15Anim."1" := #C_Config.DescriptionBit1;
       #H_GBBitShift.H_TxtInBit0_15Anim."2" := #C_Config.DescriptionBit2;
       #H_GBBitShift.H_TxtInBit0_15Anim."3" := #C_Config.DescriptionBit3;
       #H_GBBitShift.H_TxtInBit0_15Anim."4" := #C_Config.DescriptionBit4;
       #H_GBBitShift.H_TxtInBit0_15Anim."5" := #C_Config.DescriptionBit5;
       #H_GBBitShift.H_TxtInBit0_15Anim."6" := #C_Config.DescriptionBit6;
       #H_GBBitShift.H_TxtInBit0_15Anim."7" := #C_Config.DescriptionBit7;
       #H_GBBitShift.H_TxtInBit0_15Anim."8" := #C_Config.DescriptionBit8;
       #H_GBBitShift.H_TxtInBit0_15Anim."9" := #C_Config.DescriptionBit9;
       #H_GBBitShift.H_TxtInBit0_15Anim."10" := #C_Config.DescriptionBit10;
       #H_GBBitShift.H_TxtInBit0_15Anim."11" := #C_Config.DescriptionBit11;
       #H_GBBitShift.H_TxtInBit0_15Anim."12" := #C_Config.DescriptionBit12;
       #H_GBBitShift.H_TxtInBit0_15Anim."13" := #C_Config.DescriptionBit13;
       #H_GBBitShift.H_TxtInBit0_15Anim."14" := #C_Config.DescriptionBit14;
       #H_GBBitShift.H_TxtInBit0_15Anim."15" := #C_Config.DescriptionBit15;
   END_IF;
END_REGION

REGION Network 14: **** 8 - Outputs **** Shift done 1
   #O_ShiftDone1 := #Arrived1;
END_REGION

REGION Network 15: **** 8 - Outputs **** Shift done 2
   #O_ShiftDone2 := #Arrived2;
END_REGION

REGION Network 16: **** 8 - Outputs **** Shift done 3
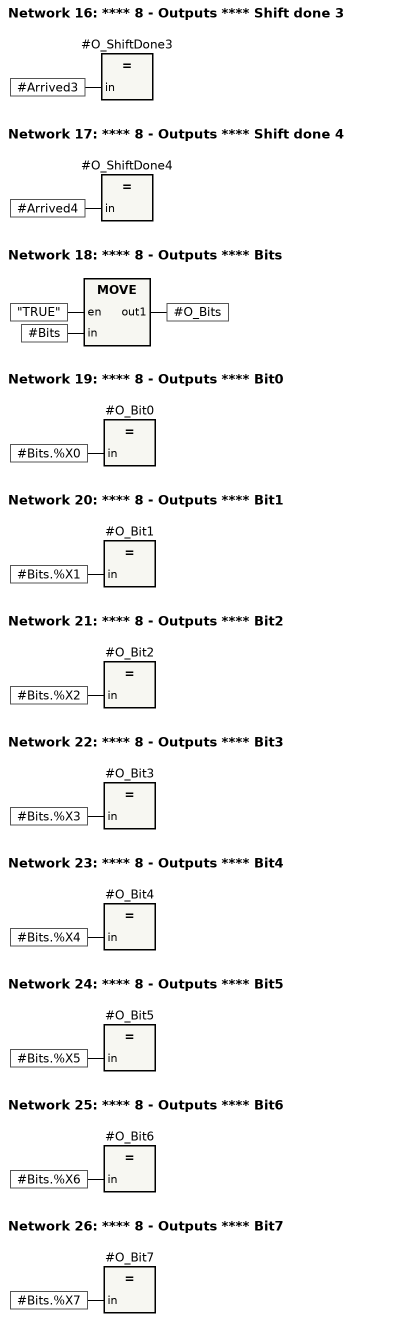
   #O_ShiftDone3 := #Arrived3;
END_REGION

REGION Network 17: **** 8 - Outputs **** Shift done 4
   #O_ShiftDone4 := #Arrived4;
END_REGION

REGION Network 18: **** 8 - Outputs **** Bits
   IF "TRUE" THEN #O_Bits := #Bits; END_IF;
END_REGION

REGION Network 19: **** 8 - Outputs **** Bit0
   #O_Bit0 := #Bits.%X0;
END_REGION

REGION Network 20: **** 8 - Outputs **** Bit1
   #O_Bit1 := #Bits.%X1;
END_REGION

REGION Network 21: **** 8 - Outputs **** Bit2
   #O_Bit2 := #Bits.%X2;
END_REGION

REGION Network 22: **** 8 - Outputs **** Bit3
   #O_Bit3 := #Bits.%X3;
END_REGION

REGION Network 23: **** 8 - Outputs **** Bit4
   #O_Bit4 := #Bits.%X4;
END_REGION

REGION Network 24: **** 8 - Outputs **** Bit5
   #O_Bit5 := #Bits.%X5;
END_REGION

REGION Network 25: **** 8 - Outputs **** Bit6
   #O_Bit6 := #Bits.%X6;
END_REGION

REGION Network 26: **** 8 - Outputs **** Bit7
   #O_Bit7 := #Bits.%X7;
END_REGION

REGION Network 27: **** 8 - Outputs **** Bit8
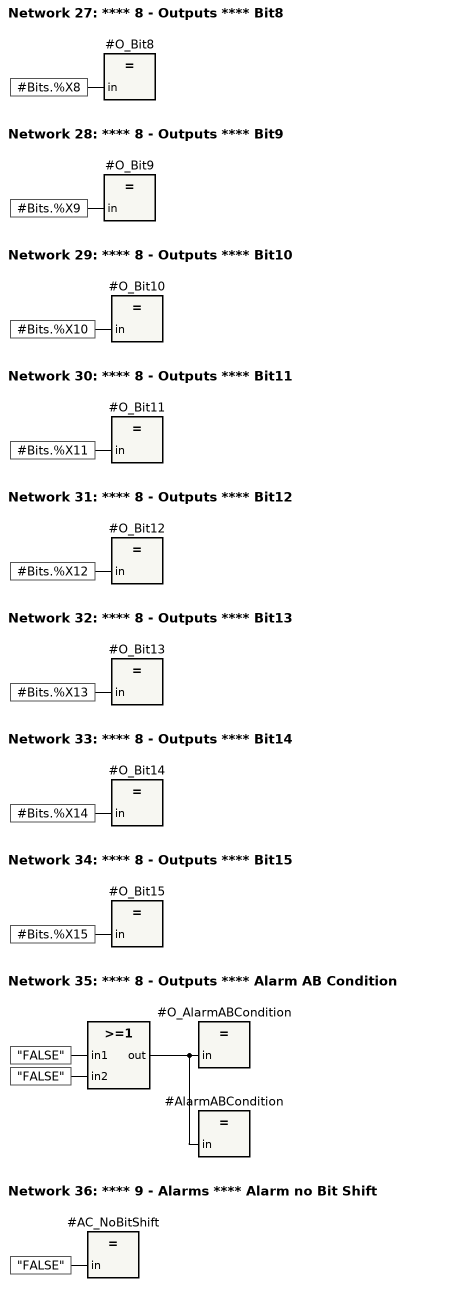
   #O_Bit8 := #Bits.%X8;
END_REGION

REGION Network 28: **** 8 - Outputs **** Bit9
   #O_Bit9 := #Bits.%X9;
END_REGION

REGION Network 29: **** 8 - Outputs **** Bit10
   #O_Bit10 := #Bits.%X10;
END_REGION

REGION Network 30: **** 8 - Outputs **** Bit11
   #O_Bit11 := #Bits.%X11;
END_REGION

REGION Network 31: **** 8 - Outputs **** Bit12
   #O_Bit12 := #Bits.%X12;
END_REGION

REGION Network 32: **** 8 - Outputs **** Bit13
   #O_Bit13 := #Bits.%X13;
END_REGION

REGION Network 33: **** 8 - Outputs **** Bit14
   #O_Bit14 := #Bits.%X14;
END_REGION

REGION Network 34: **** 8 - Outputs **** Bit15
   #O_Bit15 := #Bits.%X15;
END_REGION

REGION Network 35: **** 8 - Outputs **** Alarm AB Condition
   // Alarm AB Condition
   #O_AlarmABCondition := "FALSE" OR "FALSE";
   #AlarmABCondition := #O_AlarmABCondition;
END_REGION

REGION Network 36: **** 9 - Alarms **** Alarm no Bit Shift
   #AC_NoBitShift := "FALSE";
END_REGION

REGION Network 37: **** 9 - Alarm Summary **** Alarm A
   // Alarm A
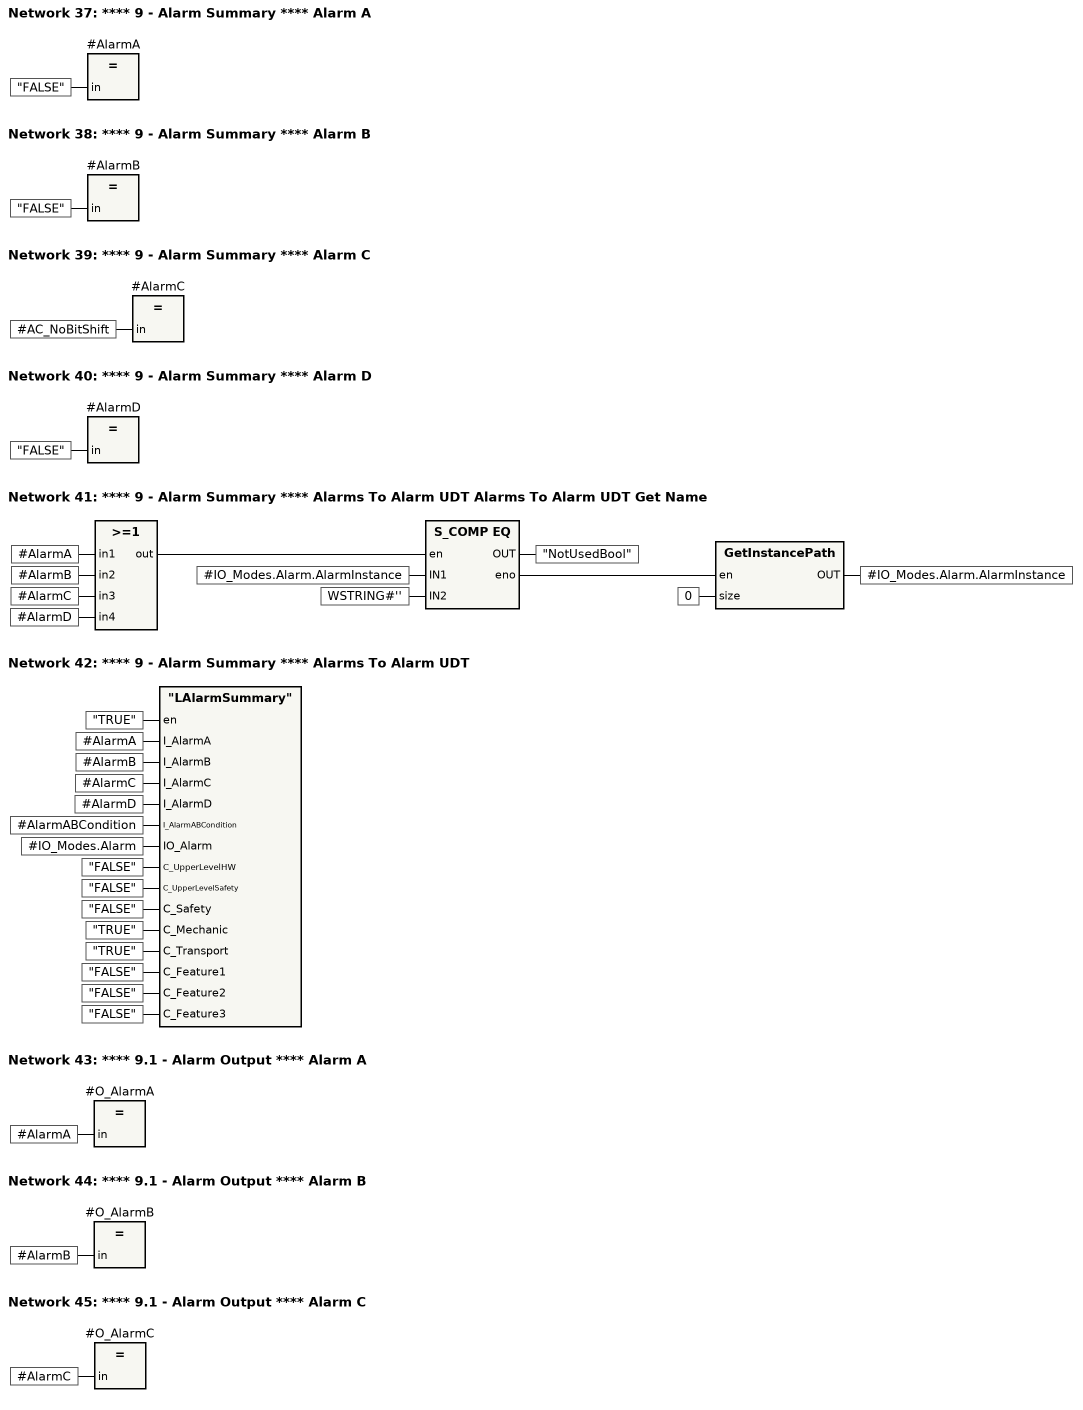
   #AlarmA := "FALSE";
END_REGION

REGION Network 38: **** 9 - Alarm Summary **** Alarm B
   // Alarm B
   #AlarmB := "FALSE";
END_REGION

REGION Network 39: **** 9 - Alarm Summary **** Alarm C
   // Alarm C
   #AlarmC := #AC_NoBitShift;
END_REGION

REGION Network 40: **** 9 - Alarm Summary **** Alarm D
   // Alarm D
   #AlarmD := "FALSE";
END_REGION

REGION Network 41: **** 9 - Alarm Summary **** Alarms To Alarm UDT Alarms To Alarm UDT Get Name
   // Alarm D
   S_COMP(EN := #AlarmA OR #AlarmB OR #AlarmC OR #AlarmD,
          IN1 := #IO_Modes.Alarm.AlarmInstance,
          IN2 := WSTRING#'',
          OUT => "NotUsedBool",
          ENO => #_w1);
   IF #_w1 THEN GetInstancePath(size := 0, OUT => #IO_Modes.Alarm.AlarmInstance); END_IF;
END_REGION

REGION Network 42: **** 9 - Alarm Summary **** Alarms To Alarm UDT
   IF "TRUE" THEN
       "LAlarmSummary"(I_AlarmA := #AlarmA,
                       I_AlarmB := #AlarmB,
                       I_AlarmC := #AlarmC,
                       I_AlarmD := #AlarmD,
                       I_AlarmABCondition := #AlarmABCondition,
                       IO_Alarm := #IO_Modes.Alarm,
                       C_UpperLevelHW := "FALSE",
                       C_UpperLevelSafety := "FALSE",
                       C_Safety := "FALSE",
                       C_Mechanic := "TRUE",
                       C_Transport := "TRUE",
                       C_Feature1 := "FALSE",
                       C_Feature2 := "FALSE",
                       C_Feature3 := "FALSE");
   END_IF;
END_REGION

REGION Network 43: **** 9.1 - Alarm Output **** Alarm A
   // Alarm A
   #O_AlarmA := #AlarmA;
END_REGION

REGION Network 44: **** 9.1 - Alarm Output **** Alarm B
   // Alarm B
   #O_AlarmB := #AlarmB;
END_REGION

REGION Network 45: **** 9.1 - Alarm Output **** Alarm C
   // Alarm C
   #O_AlarmC := #AlarmC;
END_REGION

REGION Network 46: **** 9.1 - Alarm Output **** Alarm D
   // Alarm D
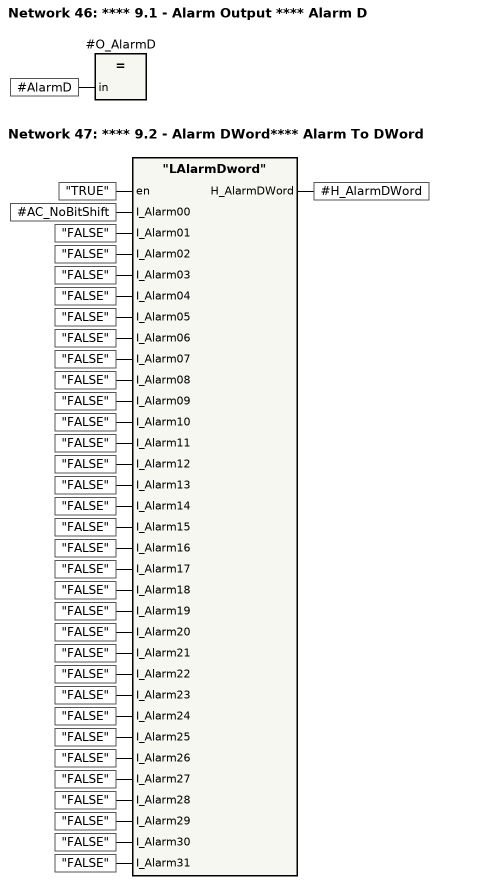
   #O_AlarmD := #AlarmD;
END_REGION

REGION Network 47: **** 9.2 - Alarm DWord**** Alarm To DWord
   // Alarm Word
   IF "TRUE" THEN
       "LAlarmDword"(I_Alarm00 := #AC_NoBitShift,
                     I_Alarm01 := "FALSE",
                     I_Alarm02 := "FALSE",
                     I_Alarm03 := "FALSE",
                     I_Alarm04 := "FALSE",
                     I_Alarm05 := "FALSE",
                     I_Alarm06 := "FALSE",
                     I_Alarm07 := "FALSE",
                     I_Alarm08 := "FALSE",
                     I_Alarm09 := "FALSE",
                     I_Alarm10 := "FALSE",
                     I_Alarm11 := "FALSE",
                     I_Alarm12 := "FALSE",
                     I_Alarm13 := "FALSE",
                     I_Alarm14 := "FALSE",
                     I_Alarm15 := "FALSE",
                     I_Alarm16 := "FALSE",
                     I_Alarm17 := "FALSE",
                     I_Alarm18 := "FALSE",
                     I_Alarm19 := "FALSE",
                     I_Alarm20 := "FALSE",
                     I_Alarm21 := "FALSE",
                     I_Alarm22 := "FALSE",
                     I_Alarm23 := "FALSE",
                     I_Alarm24 := "FALSE",
                     I_Alarm25 := "FALSE",
                     I_Alarm26 := "FALSE",
                     I_Alarm27 := "FALSE",
                     I_Alarm28 := "FALSE",
                     I_Alarm29 := "FALSE",
                     I_Alarm30 := "FALSE",
                     I_Alarm31 := "FALSE",
                     H_AlarmDWord => #H_AlarmDWord);
   END_IF;
END_REGION
END_FUNCTION_BLOCK
